FUNCTION_BLOCK FB_TelescopeErrorState EXTENDS FB_TelescopeState
VAR_INPUT
END_VAR
VAR_OUTPUT
END_VAR
VAR
END_VAR

METHOD Main : BOOL
VAR_INPUT
END_VAR
// 
// state
//

// wait until error is gone
IF NOT pMachine^.pControl^.bError THEN
	pMachine^.State := E_TelescopeState.idle;
END_IF

//
// commands
// 

IF bReset THEN
	pMachine^.pControl^.Reset();
	bReset := FALSE;
END_IF
END_METHOD

END_FUNCTION_BLOCK

(* stored: Version 1.1.0.1, ProductVersion 3.1.4024.15
   POU FB_TelescopeErrorState: Id {f6247b17-50b5-4595-95a4-537db140c4db}, SpecialFunc None
   Method Main: Id {5e502bd3-c077-408e-93cc-6a9fe7b1ce10} *)
